(* CODESYS project xlh-control-systems.library
   Author: Pascal Helfenstein - Thomas Ruoss
   Version: 0.1
   Title: xLH Control Systems
   DefaultNamespace: XlhControlSystems
   Placeholder: XlhControlSystems
   Company: xemax ag

Project tree, tasks and I/O mapping:
  libraries: Standard, 3.5.18.0 (System); VisuDialogs, * (System)
  00000000-0000-0000-0000-000000000000|D:\CoDeSys\LibrariesV3\trunk\Intern\CAA\CAA Template\3.2.0.3 draft\Prefix.pdf
  00000000-0000-0000-0000-000000000000|D:\CoDeSys\LibrariesV3\trunk\Intern\CAA\CAA Template\3.4.0.0 draft\Placeholder.xml
  00000000-0000-0000-0000-000000000000|D:\CoDeSys\LibrariesV3\trunk\Intern\CAA\CAA Template\3.5.2.0 draft\Placeholder.xml
  Library Information/
    function GetLibVersion [ST]
    function GetLibVersionNumber [ST]
    function IsLibReleased [ST]
  POUs/
    function block DT1 [ST]: reset
    data type eFiltertyp
    data type eReglertyp
    data type eSignalform
    function block I [ST]
    function block Kennlinie [ST]
    function block Limitierung [ST]
    function block Totband [ST]
    function block Logger_ [ST]
    function block P [ST]
    function block PT1 [ST]: reset
    function block PT2 [ST]: reset
    function block PT2s [ST]: reset
    function block KalmanFilter [ST]: reset
    function block PTt [ST]: reset
    function block Rauschen [ST]
    function RealToInt [ST]
    function RealToUInt [ST]
    function block Regler [ST]: Reglertyp, reset
    program CS_COMMOM [ST]
    function block Signalgenerator [ST]
    text list GlobalTextList
  text list TextListForCombobox_eReglertyp
  text list TextListForCombobox_eSignalform
  visualisation RET_VISU_Signalgenerator
  visualisation RET_VISU_Regler
  visualisation RET_VISU_I
  visualisation RET_VISU_PTt
  visualisation RET_VISU_PT2s
  visualisation RET_VISU_PT2
  visualisation RET_VISU_PT1
  visualisation RET_VISU_DT1
  visualisation RET_VISU_Rauschen
  visualisation RET_VISU_KalmanFilter
  visualisation RET_VISU_P
  visualisation RET_VISU_Limitierung
  visualisation RET_VISU_Kennlinie
  visualisation RET_VISU_Totband
  visualisation VISU_HELPER_Combobox_eReglertyp
  visualisation VISU_HELPER_Combobox_eSignalform
*)

// POUs/eFiltertyp
TYPE eFiltertyp :
(
	NONE_ := 1,
	TIEFPASS := 2,
	HOCHPASS := 3
)INT;
END_TYPE

// POUs/eReglertyp
TYPE eReglertyp :
(
	P := 1,
	I := 2,
	PI := 3,
	PDT1 := 4,
	PIDT1 := 5
)INT;
END_TYPE

// POUs/eSignalform
TYPE eSignalform :
(
	OFF := 1,
	OFFSET := 2,
	RECHTECK := 3,
	DREIECK := 4,
	SINUS := 5,
	RAMPE := 6
)INT;
END_TYPE

// Library Information/GetLibVersion
// This function has been automatically generated from the project information.
FUNCTION GetLibVersion : VERSION
VAR_INPUT
	
END_VAR

GetLibVersion.uiMajor := 0;
GetLibVersion.uiMinor := 1;
GetLibVersion.uiServicePack := 65535;
GetLibVersion.uiPatch := 65535;

END_FUNCTION

// Library Information/GetLibVersionNumber
// This function has been automatically generated from the project information.
FUNCTION GetLibVersionNumber : DWORD
VAR_INPUT
	
END_VAR

GetLibVersionNumber := 131071;

END_FUNCTION

// Library Information/IsLibReleased
// This function has been automatically generated from the project information.
FUNCTION IsLibReleased : BOOL
VAR_INPUT
	
END_VAR

IsLibReleased := FALSE;

END_FUNCTION

// POUs/DT1
{attribute 'FBVisuCreator'}
{attribute 'FBVisuCreatorPrefix' :=  'RET_VISU_'}
FUNCTION_BLOCK DT1
VAR_INPUT
	{attribute 'FBVisuCreatorFormatString' := '%1.3f'}
	rE: REAL;
	{attribute 'FBVisuCreatorFormatString' := '%1.3f'}
	rTv: REAL;
	{attribute 'FBVisuCreatorFormatString' := '%1.3f'}
	rTvz: REAL;
	{attribute 'FBVisuCreatorBoolColor' := 'Red'}
	{attribute 'FBVisuCreatorCustomName' := 'Reset'}
	bReset: BOOL;
END_VAR
VAR_OUTPUT
	{attribute 'FBVisuCreatorFormatString' := '%1.3f'}
	rA: REAL;
END_VAR
VAR
	rDxe: REAL;
	rDxa: REAL;
	rEold: REAL;
END_VAR

IF (rTvz > 0.0) THEN
	rDxe := rTv/rTvz*(rE - rEold);
	rEold := rE;
	rDxa := rA/rTvz*CS_COMMOM.rDt;
END_IF
rA := rA + rDxe - rDxa;

IF bReset THEN
	reset();
END_IF

ACTION reset:
rA := 0.0;
rEold := 0.0;
rDxe := 0.0;
rDxa := 0.0;
END_ACTION

END_FUNCTION_BLOCK

// POUs/CS_COMMOM
PROGRAM CS_COMMOM
VAR_INPUT
	rDt: REAL := 0.004;// Zykluszeit Main-Task
END_VAR

END_PROGRAM

// POUs/I
{attribute 'FBVisuCreator'}
{attribute 'FBVisuCreatorPrefix' :=  'RET_VISU_'}
FUNCTION_BLOCK I
VAR_INPUT
	{attribute 'FBVisuCreatorFormatString' := '%1.3f'}
	rX: REAL;
	{attribute 'FBVisuCreatorFormatString' := '%1.3f'}
	rTi: REAL;
	{attribute 'FBVisuCreatorBoolColor' := 'Red'}
	bReset: BOOL;
END_VAR
VAR_OUTPUT
	rY: REAL;
END_VAR
VAR
	rSumme: REAL;
END_VAR

IF (rTi > 0.0) THEN
	rSumme := rSumme + 1.0/rTi*rX*CS_COMMOM.rDt;
END_IF
IF bReset THEN
	rSumme := 0.0;
END_IF
rY := rSumme;

END_FUNCTION_BLOCK

// POUs/Kennlinie
{attribute 'FBVisuCreator'}
{attribute 'FBVisuCreatorPrefix' :=  'RET_VISU_'}
FUNCTION_BLOCK Kennlinie
VAR_INPUT
	{attribute 'FBVisuCreatorFormatString' := '%1.3f'}
	rX: REAL;
	{attribute 'FBVisuCreatorBoolColor' := 'Red'}
	{attribute 'FBVisuCreatorCustomName' := 'spiegelung an X=Y'}
	bSpiegelungXgY: BOOL := FALSE;
	{attribute 'FBVisuCreatorBoolColor' := 'Red'}
	{attribute 'FBVisuCreatorCustomName' := 'aktiviert'}
	bAktiviert: BOOL := TRUE;
	{attribute 'FBVisuCreatorExcludeEntry'}	
	arXin: ARRAY [0..10] OF REAL;
	{attribute 'FBVisuCreatorExcludeEntry'}	
	arYin: ARRAY [0..10] OF REAL;	
END_VAR
VAR_OUTPUT
	{attribute 'FBVisuCreatorFormatString' := '%1.3f'}
	rY: REAL;
END_VAR
VAR
	arX: ARRAY [0..10] OF REAL;
	arY: ARRAY [0..10] OF REAL;	
	iN: UINT;
	iI: UINT;
	rM: REAL;
	rQ: real;
	rXmin: REAL;
	rXmax: REAL;
	rYmin: REAL;
	rYmax: real;
END_VAR

IF bSpiegelungXgY THEN
	arX := arYin;
	arY := arXin;
ELSE
	arX := arXin;
	arY := arYin;
END_IF

iN := SIZEOF(arX)/4;
rXmin := arX[0];
rXmax := arX[iN- 1];
rYmin := arY[0];
rYmax := arY[iN - 1];

IF (rX <= rXmin) THEN // Überprüfung Grenzwerte Min und Max
	rY := rYmin;
ELSIF (rX >= rXmax) THEN 
	rY := rYmax;
ELSE // Eingangswert innerhalb Stützwerte
	iI := 0;
	WHILE (iI < (iN - 1)) DO
		IF (rX > arX[iI]) AND (rX <= arX[iI + 1]) THEN
			rM := (arY[iI + 1] - arY[iI])/(arX[iI + 1] - arX[iI]);
			rQ := arY[iI] - rM*arX[iI];
			rY := rM*rX + rQ;
			iI := iN;
		END_IF
		iI := iI + 1;
	END_WHILE
END_IF

IF NOT bAktiviert THEN
	rY := rX;
END_IF

(*
IF (rX < 0.01) THEN 
	rY := 0;
END_IF
*)

END_FUNCTION_BLOCK

// POUs/Limitierung
{attribute 'FBVisuCreator'}
{attribute 'FBVisuCreatorPrefix' :=  'RET_VISU_'}
FUNCTION_BLOCK Limitierung
VAR_INPUT
	{attribute 'FBVisuCreatorFormatString' := '%1.3f'}
	rY: REAL;
	{attribute 'FBVisuCreatorBoolColor' := 'Red'}
	bEnable: BOOL := TRUE;
	{attribute 'FBVisuCreatorFormatString' := '%1.3f'}
	rYmin: REAL := -10.0;
	{attribute 'FBVisuCreatorFormatString' := '%1.3f'}
	rYmax: REAL := 10.0;	
END_VAR
VAR_OUTPUT
	{attribute 'FBVisuCreatorFormatString' := '%1.3f'}
	rYlim: REAL;
	{attribute 'FBVisuCreatorBoolColor' := 'Red'}
	bAct_UL: BOOL := FALSE;
	{attribute 'FBVisuCreatorBoolColor' := 'Red'}
	bAct_LL: BOOL := FALSE;
END_VAR
VAR
	//rYmin: REAL;
	//rYmax: REAL;
END_VAR

IF bEnable THEN
	rYlim := LIMIT(rYmin, rY, rYmax);
	
	IF rY = rYlim THEN
		bAct_UL := FALSE;
		bAct_LL := FALSE;
	ELSIF rY > rYlim THEN
			bAct_UL := TRUE;
			bAct_LL := FALSE;
	ELSIF rY < rYlim THEN
		bAct_LL := TRUE;
		bAct_UL := FALSE;
	END_IF
ELSE
	rYlim := rY;
	bAct_LL := FALSE;
	bAct_UL := FALSE;
END_IF

END_FUNCTION_BLOCK

// POUs/Totband
{attribute 'FBVisuCreator'}
{attribute 'FBVisuCreatorPrefix' :=  'RET_VISU_'}
FUNCTION_BLOCK Totband
VAR_INPUT
	{attribute 'FBVisuCreatorFormatString' := '%1.3f'}
	rY: REAL;
	{attribute 'FBVisuCreatorBoolColor' := 'Red'}
	bEnable: BOOL := TRUE;
	{attribute 'FBVisuCreatorFormatString' := '%1.3f'}
	rYthreshold: REAL := 1.0;	
END_VAR
VAR_OUTPUT
	{attribute 'FBVisuCreatorFormatString' := '%1.3f'}
	rYlim: REAL;
END_VAR
VAR
	//rYmin: REAL;
	//rYmax: REAL;
END_VAR

IF bEnable THEN
	IF ABS(rY) <= rYthreshold THEN
		rYlim := 0.0;
	ELSE
		rYlim := rY;
	END_IF
ELSE
	rYlim := rY;
END_IF

END_FUNCTION_BLOCK

// POUs/Logger_
FUNCTION_BLOCK Logger_
VAR_IN_OUT
	bRunning: BOOL;
END_VAR
VAR_INPUT
	rMeasureTime: REAL := 10.0;
	uiDownsampling: UINT := 1;
	rSignal_1: REAL;
	rSignal_2: REAL;
	rSignal_3: REAL;
	rSignal_4: REAL;
	rSignal_5: REAL;
	rSignal_6: REAL;
	rSignal_7: REAL;
	rSignal_8: REAL;
	rSignal_9: REAL;
	rSignal_10: REAL;	
END_VAR
VAR_OUTPUT
	rActIndexProzent: REAL;
	arTime: ARRAY[0..999] OF REAL;
	arSignal_1: ARRAY[0..999] OF REAL;
	arSignal_2: ARRAY[0..999] OF REAL;
	arSignal_3: ARRAY[0..999] OF REAL;
	arSignal_4: ARRAY[0..999] OF REAL;
	arSignal_5: ARRAY[0..999] OF REAL;
	arSignal_6: ARRAY[0..999] OF REAL;
	arSignal_7: ARRAY[0..999] OF REAL;
	arSignal_8: ARRAY[0..999] OF REAL;
	arSignal_9: ARRAY[0..999] OF REAL;
	arSignal_10: ARRAY[0..999] OF REAL;
END_VAR
VAR
	iStateLogger: INT := 0;
	rSamplingTime: REAL;
	n: UINT;
	uiIndex: UINT;
	uiSamplingCounter: UINT;
END_VAR


// Datenlogger für die Erfassung der Sprungantwort
rSamplingTime := CS_COMMOM.rDt;
IF bRunning THEN
	IF iStateLogger = 0 THEN
		iStateLogger := 1;
	END_IF
	CASE iStateLogger OF
		0: // warte auf Sprungantwort
			//ToDo Sampling Measure time
		
		1: 	// Reset
			uiSamplingCounter := 0;
			rActIndexProzent := 0.0;
			uiIndex := 0;
			FOR n := 0 TO 999 BY 1 DO
				arTime[n] := UINT_TO_REAL(n)*CS_COMMOM.rDt*UINT_TO_REAL(uiDownsampling);
				arSignal_1[n] := 0.0;
				arSignal_2[n] := 0.0;
				arSignal_3[n] := 0.0;
				arSignal_4[n] := 0.0;
				arSignal_5[n] := 0.0;
				arSignal_6[n] := 0.0;
				arSignal_7[n] := 0.0;
				arSignal_8[n] := 0.0;
				arSignal_9[n] := 0.0;
				arSignal_10[n] := 0.0;
			END_FOR
			iStateLogger := 2;
		
		2: 
			arSignal_1[uiIndex] := rSignal_1;
			arSignal_2[uiIndex] := rSignal_2;
			arSignal_3[uiIndex] := rSignal_3;
			arSignal_4[uiIndex] := rSignal_4;
			arSignal_5[uiIndex] := rSignal_5;
			arSignal_6[uiIndex] := rSignal_6;
			arSignal_7[uiIndex] := rSignal_7;
			arSignal_8[uiIndex] := rSignal_8;
			arSignal_9[uiIndex] := rSignal_9;
			arSignal_10[uiIndex] := rSignal_10;

			rActIndexProzent := UINT_TO_REAL(uiIndex)/999.0*100.0;
		
			uiSamplingCounter := uiSamplingCounter + 1;
			IF (uiSamplingCounter >= uiDownsampling) THEN
				uiSamplingCounter := 0;
				uiIndex := uiIndex + 1;
			END_IF
			IF uiIndex >= 1000 THEN
				iStateLogger := 0;
				bRunning := FALSE;
			END_IF
		
		ELSE
			iStateLogger := 0;
			bRunning := FALSE;
	END_CASE
ELSE
	iStateLogger := 0;
END_IF

END_FUNCTION_BLOCK

// POUs/P
{attribute 'FBVisuCreator'}
{attribute 'FBVisuCreatorPrefix' :=  'RET_VISU_'}
FUNCTION_BLOCK P
VAR_INPUT
	{attribute 'FBVisuCreatorFormatString' := '%1.3f'}
	rX: REAL;
	{attribute 'FBVisuCreatorFormatString' := '%1.3f'}
	rK: REAL;
	{attribute 'FBVisuCreatorBoolColor' := 'Red'}
	bReset: BOOL;
END_VAR
VAR_OUTPUT
	rY: REAL;
END_VAR
VAR
	rSumme: REAL;
END_VAR

rY := rX*rK;
IF bReset THEN
	rY := 0.0;
END_IF

END_FUNCTION_BLOCK

// POUs/PT1
{attribute 'FBVisuCreator'}
{attribute 'FBVisuCreatorPrefix' :=  'RET_VISU_'}
FUNCTION_BLOCK PT1
VAR_INPUT
	{attribute 'FBVisuCreatorFormatString' := '%1.3f'}	
	rX: REAL;
	{attribute 'FBVisuCreatorFormatString' := '%1.3f'}
	rK: REAL;
	{attribute 'FBVisuCreatorFormatString' := '%1.3f'}
	rT: REAL;
	{attribute 'FBVisuCreatorBoolColor' := 'Red'}
	{attribute 'FBVisuCreatorCustomName' := 'Reset'}
	bReset: BOOL;
END_VAR
VAR_OUTPUT
	{attribute 'FBVisuCreatorFormatString' := '%1.3f'}
	rY: REAL;
END_VAR
VAR
	rSumme: REAL;
END_VAR

IF bReset THEN
	reset();
END_IF

IF (rT > 0.0) THEN
	rY := rY + (-rY + rK*rX)/MAX(rT,0.001)*CS_COMMOM.rDt;
ELSE
	rY := rX;
END_IF

ACTION reset:
rY := 0.0;
END_ACTION

END_FUNCTION_BLOCK

// POUs/PT2
{attribute 'FBVisuCreator'}
{attribute 'FBVisuCreatorPrefix' :=  'RET_VISU_'}
FUNCTION_BLOCK PUBLIC PT2
VAR_INPUT
	{attribute 'FBVisuCreatorFormatString' := '%1.3f'}
	rX: REAL;
	{attribute 'FBVisuCreatorFormatString' := '%1.3f'}
	rK: REAL;
	{attribute 'FBVisuCreatorFormatString' := '%1.3f'}
	rT1: REAL;
	{attribute 'FBVisuCreatorFormatString' := '%1.3f'}
	rT2: REAL;
	{attribute 'FBVisuCreatorBoolColor' := 'Red'}
	{attribute 'FBVisuCreatorCustomName' := 'Reset'}
	bReset: BOOL;
END_VAR
VAR_OUTPUT
	{attribute 'FBVisuCreatorFormatString' := '%1.3f'}
	rY: REAL;
END_VAR
VAR 
	rZeta: REAL;
	rOmega: REAL;
	rXX: REAL;
	rDx: REAL;
	rDy: REAL;
END_VAR

// Umrechnung der Faktoren in PT2s
rOmega := 1/SQRT(MAX(rT1*rT2, 0.001));
rZeta := rOmega*(rT1+rT2)/2.0;

IF bReset THEN
	reset();
END_IF

rDy := CS_COMMOM.rDt*rOmega*rXX;
rDx := CS_COMMOM.rDt*rOmega*(rK*rX - rY - 2*rZeta*rXX);
rXX := rXX + rDx;
rY := rY + rDy;

ACTION reset:
rXX := 0.0;
rY := 0.0;
END_ACTION

END_FUNCTION_BLOCK

// POUs/PT2s
{attribute 'FBVisuCreator'}
{attribute 'FBVisuCreatorPrefix' :=  'RET_VISU_'}
FUNCTION_BLOCK PUBLIC PT2s
VAR_INPUT
	{attribute 'FBVisuCreatorFormatString' := '%1.3f'}
	rX: REAL;
	{attribute 'FBVisuCreatorFormatString' := '%1.3f'}
	rK: REAL;
	{attribute 'FBVisuCreatorFormatString' := '%1.3f'}
	rZeta: REAL;
	{attribute 'FBVisuCreatorFormatString' := '%1.3f'}
	rOmega: REAL;
	{attribute 'FBVisuCreatorBoolColor' := 'Red'}
	{attribute 'FBVisuCreatorCustomName' := 'Reset'}
	bReset: BOOL;
END_VAR
VAR_OUTPUT
	{attribute 'FBVisuCreatorFormatString' := '%1.3f'}
	rY: REAL;
END_VAR
VAR 
	rXX: REAL;
	rDx: REAL;
	rDy: REAL;
END_VAR

rDy := CS_COMMOM.rDt*rOmega*rXX;
rDx := CS_COMMOM.rDt*rOmega*(rK*rX - rY - 2*rZeta*rXX);
rXX := rXX + rDx;
rY := rY + rDy;

IF bReset THEN
	reset();
END_IF

ACTION reset:
rXX := 0.0;
rY := 0.0;
END_ACTION

END_FUNCTION_BLOCK

// POUs/KalmanFilter
{attribute 'FBVisuCreator'}
{attribute 'FBVisuCreatorPrefix' :=  'RET_VISU_'}
FUNCTION_BLOCK PUBLIC KalmanFilter
VAR_INPUT
	{attribute 'FBVisuCreatorFormatString' := '%1.3f'}
	rX: REAL;
	{attribute 'FBVisuCreatorFormatString' := '%1.3f'}
	rQ: REAL;
	{attribute 'FBVisuCreatorFormatString' := '%1.3f'}
	rR: REAL;
	{attribute 'FBVisuCreatorCustomName' := 'Reset'}
	bReset: BOOL;
END_VAR
VAR_OUTPUT
	{attribute 'FBVisuCreatorFormatString' := '%1.3f'}
	rY: REAL;
END_VAR
VAR 
	X_hat: REAL;
	X_hat_min: REAL;
	poise: REAL;
	Pmin: REAL;
	K: REAL;
	rAvoidZero: REAL := 0.001;
END_VAR


IF bReset THEN
	reset();
END_IF

K := Pmin/MAX((Pmin + rR), rAvoidZero);
X_hat := X_hat_min + K*(rX - X_hat_min);
poise := (1 - K)*Pmin;
Pmin := poise + rQ;
X_hat_min := X_hat;
rY := X_hat;

ACTION reset:
X_hat := 0.0;
X_hat_min := 0.0;
poise := 0.0;
Pmin := 0.0;
K := 0.0;
rY := 0.0;
END_ACTION

END_FUNCTION_BLOCK

// POUs/PTt
{attribute 'FBVisuCreator'}
{attribute 'FBVisuCreatorPrefix' :=  'RET_VISU_'}
FUNCTION_BLOCK PUBLIC PTt
VAR_INPUT
	{attribute 'FBVisuCreatorFormatString' := '%1.3f'}
	rX: REAL;
	{attribute 'FBVisuCreatorFormatString' := '%1.3f'}
	rK: REAL := 1.0;
	{attribute 'FBVisuCreatorFormatString' := '%1.3f'}
	rTt: REAL;
	{attribute 'FBVisuCreatorBoolColor' := 'Red'}
	{attribute 'FBVisuCreatorCustomName' := 'Reset'}
	bReset: BOOL;
END_VAR
VAR_OUTPUT
	{attribute 'FBVisuCreatorFormatString' := '%1.3f'}
	rY: REAL;
END_VAR
VAR 
	arX: ARRAY [0..5000] OF REAL;
	iN: INT;
	ii: INT;
END_VAR

IF bReset THEN
	rTt := CS_COMMOM.rDt;
	reset();
END_IF

iN := REAL_TO_INT(rTt/MAX(CS_COMMOM.rDt, 0.001));
iN := LIMIT(1, iN, 5000);
FOR ii := iN TO 1 BY -1 DO
	arX[ii] := arX[ii - 1];
END_FOR
arX[0] := rX;
rY := rK*arX[iN];

ACTION reset:
rY := 0.0;
END_ACTION

END_FUNCTION_BLOCK

// POUs/Rauschen
{attribute 'FBVisuCreator'}
{attribute 'FBVisuCreatorPrefix' :=  'RET_VISU_'}
FUNCTION_BLOCK Rauschen
VAR_INPUT
	{attribute 'FBVisuCreatorFormatString' := '%1.3f'}
	rVerstaerkung: REAL;
END_VAR
VAR_OUTPUT
	{attribute 'FBVisuCreatorFormatString' := '%1.3f'}
	rY: REAL;
END_VAR
VAR
	rSumme: REAL;
	iI: INT := 0;
END_VAR
VAR CONSTANT
	// Array mit Zufallszahlen in einem Bereich 0.0 <= rnd < 1.0
